TYPE DUT_AmpelConfig :
STRUCT
	tRot		:TIME; // Zet für die Rotphase
	tRotGelb	:TIME;	// Zeit für die RotGruenphase
	tGruen		:TIME;	// Zeit für die Gruenpahse
	tGelb		:TIME;	// Zeit für die Gelbphase
	active		: BOOL;
END_STRUCT
END_TYPE

(* stored: Version 1.1.0.1, ProductVersion 3.1.4024.12
   DUT DUT_AmpelConfig: Id {5b2e8a0d-668f-46f3-a2ce-a0703933cda9} *)
